FUNCTION_BLOCK FB_LamparaIntermitente_SFC_2
VAR_INPUT
    TiempoParpadeo: REAL := 0.5;
END_VAR
VAR_OUTPUT
END_VAR
VAR
    Lampara AT %Q*: BOOL;
END_VAR

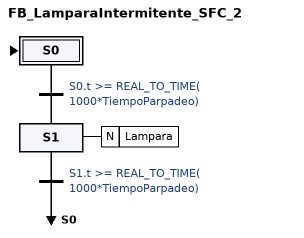
INITIAL_STEP S0:
END_STEP
TRANSITION FROM S0 TO S1
    := S0.t >= REAL_TO_TIME(1000*TiempoParpadeo);
END_TRANSITION
STEP S1:
    Lampara(N);
END_STEP
TRANSITION FROM S1 TO S0
    := S1.t >= REAL_TO_TIME(1000*TiempoParpadeo);
END_TRANSITION

END_FUNCTION_BLOCK

(* stored: Version 1.1.0.1, ProductVersion 3.1.4024.15
   POU FB_LamparaIntermitente_SFC_2: Id {60a9ce2c-efe0-44ed-bd4f-aa8838fb79b1}, SpecialFunc None *)
